VAR_GLOBAL
	fbSaftey:		FB_Component;	
END_VAR

(* stored: Version 1.1.0.1, ProductVersion 3.1.4024.12
   GVL GVL: Id {d2c8887b-6ecf-48d3-87de-d7040ac613e3} *)
